DATA_BLOCK "Retain_DB"
{ S7_Optimized_Access := 'TRUE' }
AUTHOR : Searinox
VERSION : 0.1
NON_RETAIN
   VAR RETAIN
      Settings : Struct
         MaxPressureDeltaPerc1 { S7_SetPoint := 'True'} : Real;   // Maximum pressure difference in percent before error
         MaxPressureDeltaPerc2 { S7_SetPoint := 'True'} : Real;   // Maximum pressure difference in percent before error
         MaxTempTransgression { S7_SetPoint := 'True'} : Real;   // Maximum temperature overrun of setpoint in centigrade before error
         SprayPipeOpenTimeout { S7_SetPoint := 'True'} : Time;   // Maximum time until spray tube must be open before error
         SetPointTempPlant : Real;
         SetPointTempFurnace : Real;
         SurgeTankLevel : Struct
            RunDry { S7_SetPoint := 'True'} : Int;   // position 4, e.g. minimum value reached
            SetPointLower { S7_SetPoint := 'True'} : Int;   // position 3, e.g. lower preset value reached
            SetPointUpper { S7_SetPoint := 'True'} : Int;   // position 2, e.g. upper preset value reached
            Overflow { S7_SetPoint := 'True'} : Int;   // position 1, e.g. maximum value reached
         END_STRUCT;
      END_STRUCT;
   END_VAR


BEGIN
   Settings.MaxPressureDeltaPerc1 := 50.0;
   Settings.MaxPressureDeltaPerc2 := 50.0;
   Settings.MaxTempTransgression := 4.0;
   Settings.SprayPipeOpenTimeout := T#15s;
   Settings.SetPointTempPlant := 27.0;
   Settings.SetPointTempFurnace := 27.0;
   Settings.SurgeTankLevel.RunDry := 2;
   Settings.SurgeTankLevel.SetPointLower := 4;
   Settings.SurgeTankLevel.SetPointUpper := 6;
   Settings.SurgeTankLevel.Overflow := 14;

END_DATA_BLOCK

